	        DefProcChngOrig:
	            //================================== Traitement des reponses pour le defaut1  =============================================================//
	            IF #ChPont.Dial_Def.Reponse_Def = 'ABANDON' THEN
	                #ChPont.Dial_Def.Reponse_Def := '';
	                IF #ChPont._Commande._PtcelOrig._Moborg <> -1 AND #ChPont._Commande._PtcelOrig._Moborg <> "Index_Mobile"(#ChPont._ChargCommun.CntlDest.Dest) THEN
	                    #ChPont._ChargCommun._VidCirChgCell := TRUE;
	                END_IF;
	                #Ret_int := "RechIndexCel"(#ChPont._ChargCommun.CntlDest.Dest);
	                #ChPont._Commande._PtcelOrig := "DB_Mod_Cellule"._TabCel[#Ret_int];
	                IF #ChPont._ChargCommun._VidCirChgCell THEN
	                    #ChPont._SuspCircuit := FALSE;
	                    #ChPont._ChargCommun._CommunGeneral._Etp := #Etape_VidCircuit;
	                    RETURN;
	                ELSE
	                    #ChPont._ChargCommun._CommunGeneral._Etp := #Etape_CtrlColChute;
	                    RETURN;
	                END_IF;
	                RETURN;
	            END_IF;
	            IF #ChPont.Dial_Def.Reponse_Def = 'RELANCE' THEN
	                #ret_string := "Proc_ChangOrig"(NumPoste := "Num_Poste",
	                                                IdComLign := #ChPont._Commande._IdComLig,
	                                                IdLigOrig := #ChPont._Commande._IdLigOrig,
	                                                NvOrig := #ChPont._ChargCommun.CntlDest.Dest,
	                                                ChgAuto := 'N',
	                                                Msg_Def => #Mess_Def, ComLign := #ChPont._Commande);
	                IF #ret_string = 'NOK' THEN
	                    #ChPont.Dial_Def.Reponse_Def := '';
	                    #Text_Def := #Mess_Def;
	                    #ChPont._ParamTrouve := FALSE;
	                    #ChPont.Dial_Def.Num_Def_Etape := 3;
	                    #ChPont.Dial_Def.Index_Defaut := "Dialog_Defaut"(Fg_Base := #FgBase,
	                                                                     Msg_Defaut := #Text_Def,
	                                                                     Type_Defaut := 2,
	                                                                     Automatisme := #ChPont._ChargCommun._CommunGeneral._Autom,
	                                                                     Num_Lot := #ChPont._ChargCommun._CommunGeneral._NumLot,
	                                                                     Origine_Defaut := 'Proc Chngm Orig',
	                                                                     Libelle_Origine := 'Changement Origine',
	                                                                     Acq1 := 'ABANDON',
	                                                                     Acq2 := 'RELANCE',
	                                                                     Acq3 := '',
	                                                                     Acq4 := '',
	                                                                     Acq5 := '',
	                                                                     Acq6 := '',
	                                                                     Acq7 := '',
	                                                                     Acq8 := '',
	                                                                     Acq_Choisi := -1,
	                                                                     Date_Arrivee := #ChPont._TpsPicke);
	                    #ChPont._ChargCommun._CommunGeneral._Etp := #Etape_Attente_RepDial;
	                    RETURN;
	                ELSE
	                    IF #ChPont._Commande._PtcelOrig._Moborg <> -1 AND #ChPont._Commande._PtcelOrig._Moborg <> "Index_Mobile"(#ChPont._ChargCommun.CntlDest.Dest) THEN
	                        #ChPont._ChargCommun._VidCirChgCell := TRUE;
	                    END_IF;
	                    #Ret_int := "RechIndexCel"(#ChPont._ChargCommun.CntlDest.Dest);
	                    #ChPont._Commande._PtcelOrig := "DB_Mod_Cellule"._TabCel[#Ret_int];
	                    IF #ChPont._ChargCommun._VidCirChgCell THEN
	                        #ChPont._SuspCircuit := FALSE;
	                        #ChPont._ChargCommun._CommunGeneral._Etp := #Etape_VidCircuit;
	                        RETURN;
	                    ELSE
	                        #ChPont._ChargCommun._CommunGeneral._Etp := #Etape_CtrlColChute;
	                        RETURN;
	                    END_IF;
	                END_IF;
	            END_IF;
	            //============================================  Fin traitement  ====================================================================//







	        END_REGION Traitement cyclique "DefArrProd"
	(*
	 *************************************** *************************************** *************************************** *************************************** ***************************************
	                                                        ╔════════════════════════════════════╗
	                                                        ║          Etape "SuspChgtCase"      ║
	                                                        ╚════════════════════════════════════╝
	*************************************** *************************************** *************************************** *************************************** ***************************************
	*)
	    #Etape_SuspChgtCase:
	        REGION Traitement preliminaire "SuspChgtCase"
	            IF (#ChPont._ChargCommun._CommunGeneral._Etp <> #ChPont._ChargCommun._CommunGeneral._EtpPrec) THEN
	                #ChPont._ChargCommun._CommunGeneral._EtpPrec := #ChPont._ChargCommun._CommunGeneral._Etp;
	                #ChPont._ChargCommun._CommunGeneral._DescEtp := 'Etape SuspChgtCase';
	                "MajBtSupervChPont"(Type := 3,
	                                    ChPont := #ChPont);
	                #ChPont._MemoAppuiBP := 0;
	            END_IF;
	        END_REGION Traitement preliminaire
	        REGION Traitement cyclique "SuspChgtCase"

	            IF #ChPont._ChargDebit THEN
	                "SuspCalculDebit"(Type := "BTSUSP",
	                                  ParCal := #ChPont._ChargCommun._CommunGeneral._ParCal);
	            END_IF;
	            IF #ChPont._Commande._Case < #ChPont._Commande._NbCase - 1 AND #ChPont._DemChgtCase = 0 THEN
	                #ChPont._IndexTemp := #ChPont._Commande._Case + 1;
	                "MemoPoidsCase"(IndexNouvCase := #ChPont._IndexTemp,
	                                Chpont := #ChPont);

	            ELSIF #ChPont._DemChgtCase <> 0 THEN
	                #ChPont._IndexTemp := #ChPont._DemChgtCase;
	                "MemoPoidsCase"(IndexNouvCase := #ChPont._IndexTemp,
	                                Chpont := #ChPont);
	                #ChPont._DemChgtCase := 0;

	            ELSE
	                //Affiche mssg def: Quantite case camion atteinte, veuillez choisir une nouvelle case
	                //Selection parmi  pt_zs->Cases[i].noCase
	                ;
	            END_IF;
	            #ChPont._ChargCommun._PtAff._MessOper := 'Attente positionnement camion et DepCycle ou FinChar pour vidanger';
	            #ChPont._ChargCommun._PtAff._NumCaseEc := #ChPont._Commande._Case;
	            #ChPont._DemChgtCase := 0;
	            #ChPont._Bouton := "LireActionBoutonChPont"(#ChPont);
	            IF #ChPont._Bouton = "DEBCYCLE" THEN
	                #ChPont._BtDepCycle := 1;
	                #ChPont._MemoAppuiBP := 0;
	                IF "CondChargement"(#ChPont) AND "FC_Test_Niv_AmontAval"(Num_Zone := #ChPont._ChargCommun._CommunGeneral._NumZone, Lst_Taches := #ChPont._ListeTaAttAutDemarrage) THEN
	                    #ChPont._SuspCircuit := FALSE;
	                    IF #ChPont._ChargDebit THEN
	                        "SuspCalculDebit"(Type := "DEBCYCLE",
	                                          ParCal := #ChPont._ChargCommun._CommunGeneral._ParCal);
	                    END_IF;
	                    #ChPont._ChargCommun._CommunGeneral._Etp := #Etape_Extract;
	                    RETURN;
	                END_IF;
	            END_IF;

	            IF #ChPont._Bouton = "ABANDONCHARG" THEN
	                #ChPont._SuspCircuit := FALSE;
	                #ChPont._Ptzs._FgStopMiPesee := FALSE;
	                #ChPont._ChargCommun._CommunGeneral._Etp := #Etape_VidCircuit;
	                RETURN;
	            END_IF;
	            "ControleChgtCase"(#ChPont);



	        END_REGION Traitement cyclique "SuspChgtCase"
	    (*
	    *************************************** *************************************** *************************************** *************************************** ***************************************
	                                                        ╔════════════════════════════════════╗
	                                                        ║          Etape "SuspChargement"    ║
	                                                        ╚════════════════════════════════════╝
	    *************************************** *************************************** *************************************** *************************************** ***************************************
	    *)
	    #Etape_SuspChargement:
	        REGION Traitement preliminaire "SuspChargement"
	            IF (#ChPont._ChargCommun._CommunGeneral._Etp <> #ChPont._ChargCommun._CommunGeneral._EtpPrec) THEN
	                #ChPont._ChargCommun._CommunGeneral._EtpPrec := #ChPont._ChargCommun._CommunGeneral._Etp;
	                #ChPont._ChargCommun._CommunGeneral._DescEtp := 'Etape SuspChargement';
	                //Suspension calcul debit
	                IF #ChPont._ChargDebit THEN
	                    "SuspCalculDebit"(Type := "BTSUSP",
	                                      ParCal := #ChPont._ChargCommun._CommunGeneral._ParCal);
	                END_IF;
	                "MajBtSupervChPont"(Type := 3,
	                                    ChPont := #ChPont);
	                #ChPont._ChargCommun._PtAff._MessOper := 'Suspension chargement';
	            END_IF;
	        END_REGION Traitement preliminaire
	        REGION Traitement cyclique "SuspChargement"
	            #ChPont._Bouton := "LireActionBoutonChPont"(#ChPont);
	            IF #ChPont._Commande._FgaVider THEN
	                IF #ChPont._ChargCommun._BpVide THEN
	                    #ChPont._Ptzs._TypeArret := "ARRET_VIDE";
	                    #ChPont._AutorMAJColChute := FALSE;
	                    #ChPont._ChargCommun._CommunGeneral._Etp := #Etape_VidCircuit;
	                    RETURN;
	                END_IF;
	            END_IF;
	            IF "CondChargement"(#ChPont) AND #ChPont._Bouton = "DEBCYCLE" THEN
	                #ChPont._SuspCircuit := FALSE;
	                IF #ChPont._ChargDebit THEN
	                    "SuspCalculDebit"(Type := "DEBCYCLE",
	                                      ParCal := #ChPont._ChargCommun._CommunGeneral._ParCal);
	                END_IF;
	                #ChPont._ChargCommun._CommunGeneral._Etp := #Etape_Extract;
	                RETURN;
	            END_IF;
	            IF #ChPont._Bouton = "ABANDONCHARG" THEN
	                IF #ChPont._ArrImmMemeProd AND #ChPont._Ptzs._FgDemArrImm THEN
	                    #ChPont._SuspCircuit := FALSE;
	                    #ChPont._Ptzs._TypeArret := "ARRET_IMM";
	                ELSE
	                    #ChPont._SuspCircuit := FALSE;
	                END_IF;
	                #ChPont._Ptzs._FgStopMiPesee := FALSE;
	                #ChPont._ChargCommun._CommunGeneral._Etp := #Etape_VidCircuit;
	                RETURN;
	            END_IF;

	            // Demande de changement de case
	            IF #ChPont._DemChgtCase <> 0 THEN
	                #ChPont._DemVib := FALSE;
	                "ArretVibreur"(#ChPont._Commande._PtcelOrig);
	                #ChPont._SuspCircuit := TRUE;
	                "Arret_Ext"(ConsQte := #ChPont._Commande._ConsQteTot,
	                            Commande := #ChPont._Commande,
	                            ChargCommun := #ChPont._ChargCommun,
	                            Ptcel := #ChPont._Commande._PtcelOrig);
	                #ChPont._ChargCommun._PtAff._ExtEc := 0;
	                #ChPont._ChargCommun._CommunGeneral._Etp := #Etape_SuspChgtCase;
	                RETURN;
	            END_IF;


	        END_REGION Traitement cyclique "SuspChargement"
	    (*
	    *************************************** *************************************** *************************************** *************************************** ***************************************
	                                                        ╔════════════════════════════════════╗
	                                                        ║      Etape "ConfFinChargement"     ║
	                                                        ╚════════════════════════════════════╝
	    *************************************** *************************************** *************************************** *************************************** ***************************************
	    *)
	    #Etape_ConfFinChargement:
	        REGION Traitement preliminaire "ConfFinChargement"
	            IF (#ChPont._ChargCommun._CommunGeneral._Etp <> #ChPont._ChargCommun._CommunGeneral._EtpPrec) THEN
	                #ChPont._ChargCommun._CommunGeneral._EtpPrec := #ChPont._ChargCommun._CommunGeneral._Etp;
	                #ChPont._ChargCommun._CommunGeneral._DescEtp := 'Etape ConfFinChargement';
	                #MajNiv := "Maj_Niv"(Num_Zone := #ChPont._ChargCommun._CommunGeneral._NumZone, Num_Tache := #ChPont._ChargCommun._CommunGeneral._Tache, Niveau := "NIV_SURPONT_CONF_FIN_CHAR");
	                #ChPont._ChargCommun._DemVibrCel := FALSE;
	                "ArretVibreur"(#ChPont._Commande._PtcelOrig);
	                #ChPont._SuspCircuit := TRUE;
	                "Arret_Ext"(ConsQte := #ChPont._Commande._ConsQteTot,
	                            Commande := #ChPont._Commande,
	                            ChargCommun := #ChPont._ChargCommun,
	                            Ptcel := #ChPont._Commande._PtcelOrig);





	                // si stop mi pesee pas de confirmation fin
	                IF #ChPont._Ptzs._FgStopMiPesee THEN
	                    #ChPont._ChargCommun._CommunGeneral._Etp := #Etape_VidCircuit;
	                    RETURN;
	                END_IF;
	                "ArretCalculDebit"(#ChPont._ChargCommun._CommunGeneral._ParCal);
	                "MajBtSupervChPont"(Type := 4,
	                                    ChPont := #ChPont);
	                IF NOT #ChPont._Ptzs._HorsPont THEN
	                    #ChPont._ChargCommun._PtAff._MessOper := 'Attente Confirmation Fin Chargement ou Ajout';
	                ELSE
	                    #ChPont._ChargCommun._PtAff._MessOper := 'Attente Camion sur pont et Confirmation Fin Chargement ou Ajout';
	                END_IF;

	                #ChPont._MemoRajout := FALSE;


	            END_IF;
	        END_REGION Traitement preliminaire
	        REGION Traitement cyclique "ConfFinChargement"
	            // On controle le changement de case dans le cas o on utilisait le bouton AJOUT
	            IF #ChPont._GestQteCaseAuto AND NOT #ChPont._Ptzs._Cases[#ChPont._Commande._Case]._FgRelCharge AND #ChPont._Commande._NbCase > 1 THEN

	                IF #ChPont._Commande._PtcelOrig._FgColChuteChgtCase = 1 THEN
	                    #ChPont._ChargCommun._QteCase := #ChPont._Ptzs._Cases[#ChPont._Commande._Case]._QteDejaChargee + #ChPont._ChargCommun._Vbasc - #ChPont._Ptzs._Cases[#ChPont._Commande._Case]._Tare + #ChPont._Commande._ChuteCel;
	                ELSIF #ChPont._Commande._PtcelOrig._FgColChuteChgtCase = 2 THEN
	                    #ChPont._ChargCommun._QteCase := #ChPont._Ptzs._Cases[#ChPont._Commande._Case]._QteDejaChargee + #ChPont._ChargCommun._Vbasc - #ChPont._Ptzs._Cases[#ChPont._Commande._Case]._Tare + #ChPont._ChuteArrImm;
	                ELSE
	                    #ChPont._ChargCommun._QteCase := #ChPont._Ptzs._Cases[#ChPont._Commande._Case]._QteDejaChargee + #ChPont._ChargCommun._Vbasc - #ChPont._Ptzs._Cases[#ChPont._Commande._Case]._Tare;
	                END_IF;

	                IF #ChPont._Ptzs._Cases[#ChPont._Commande._Case]._ConsQte > 0 AND ((#ChPont._ChargCommun._QteCase > #ChPont._Ptzs._Cases[#ChPont._Commande._Case]._ConsQte + #ChPont._TolDernCase AND #ChPont._Commande._Case = #ChPont._Commande._NbCase - 1) OR
	                    (#ChPont._ChargCommun._QteCase > #ChPont._Ptzs._Cases[#ChPont._Commande._Case]._ConsQte AND #ChPont._Commande._Case <> #ChPont._Commande._NbCase - 1)) THEN

	                    #ChPont._ChargCommun._DemVibrCel := FALSE;
	                    "ArretVibreur"(#ChPont._Commande._PtcelOrig);
	                    #ChPont._SuspCircuit := TRUE;
	                    "Arret_Ext"(ConsQte := #ChPont._Commande._ConsQteTot,
	                                Commande := #ChPont._Commande,
	                                ChargCommun := #ChPont._ChargCommun,
	                                Ptcel := #ChPont._Commande._PtcelOrig);
	                    #ChPont._Ptzs._Cases[#ChPont._Commande._Case]._FgRelCharge := TRUE;
	                    #ChPont._ChargCommun._PtAff._ExtEc := 0;
	                    #ChPont._ChargCommun._CommunGeneral._Etp := #Etape_SuspChgtCase;
	                    RETURN;
	                END_IF;
	            END_IF;

	            #ChPont._Bouton := "LireActionBoutonChPont"(#ChPont);
	            IF #ChPont._Bouton = "BTAJOUT" THEN
	                #ChPont._SuspCircuit := FALSE;
	                #ChPont._MemoRajout := TRUE;
	                #ChPont._AutorMAJColChute := FALSE;
	                #ChPont._ChargCommun._CommunGeneral._Etp := #Etape_Extract;         // #Etape_Surveillance;
	                RETURN;
	            END_IF;
	            IF #ChPont._Bouton = "ABANDONCHARG" OR #ChPont._VidAuto THEN
	                // Redemarrage circuit si pas arret immdiat
	                IF #ChPont._Ptzs._TypeArret <> "ARRET_IMM" THEN
	                    #ChPont._SuspCircuit := FALSE;
	                END_IF;
	                #ChPont._ChargCommun._CommunGeneral._Etp := #Etape_VidCircuit;
	                RETURN;
	            END_IF;
	            IF #ChPont._Bouton = "BTSUSP" THEN
	                #ChPont._BtSusp := 1;
	                #ChPont._MemoAppuiBP := 0;
	                #ChPont._SuspCircuit := TRUE;
	                #Ret_RD_Sys_T := RD_SYS_T(#ChPont._DebFermExt);
	            END_IF;
	        END_REGION Traitement cyclique "ConfFinChargement"
	    (*
	    *************************************** *************************************** *************************************** *************************************** ***************************************
	                                                        ╔════════════════════════════════════╗
	                                                        ║          Etape "VidCircuit"        ║
	                                                        ╚════════════════════════════════════╝
	    *************************************** *************************************** *************************************** *************************************** ***************************************
	    *)
	    #Etape_VidCircuit:
	        REGION Traitement preliminaire "VidCircuit"
	            IF (#ChPont._ChargCommun._CommunGeneral._Etp <> #ChPont._ChargCommun._CommunGeneral._EtpPrec) THEN
	                #ChPont._ChargCommun._CommunGeneral._EtpPrec := #ChPont._ChargCommun._CommunGeneral._Etp;
	                #ChPont._ChargCommun._CommunGeneral._DescEtp := 'Etape VidCircuit';
	                #MajNiv := "Maj_Niv"(Num_Zone := #ChPont._ChargCommun._CommunGeneral._NumZone, Num_Tache := #ChPont._ChargCommun._CommunGeneral._Tache, Niveau := "NIV_SURPONT_VID_CIR");
	                #ChPont._ChargCommun._PtAff._MessOper := 'Vidange circuit';
	                "ArretCalculDebit"(#ChPont._ChargCommun._CommunGeneral._ParCal);
	                "Arret_Ext"(ConsQte := #ChPont._Commande._ConsQteTot,
	                            Commande := #ChPont._Commande,
	                            ChargCommun := #ChPont._ChargCommun,
	                            Ptcel := #ChPont._Commande._PtcelOrig);
	                // fonction utilisateur avant vidange circuit
	                IF #ChPont._ActionAvantVidangeCircuit THEN
	                    "ActionAvantVidangeCircuit"();
	                END_IF;
	                // Vidange cellule sur changement de cellule
	                (*  IF #ChPont._ChargCommun._VidCirChgCell THEN
	    #ChPont._ChargCommun._DefEvol := 0;
	    #ChPont._ChargCommun._CommunGeneral._Etp := #Etape_CtrlColChute;
	    #ChPont._ChargCommun._VidCirChgCell := FALSE;
	    RETURN;
	    END_IF; *)
	            END_IF;
	        END_REGION Traitement preliminaire
	        REGION Traitement cyclique "VidCircuit"
	            #ChPont._Bouton := "LireActionBoutonChPont"(#ChPont);
	            IF #ChPont._Bouton = "BTSUSP" THEN
	                #ChPont._BtSusp := 1;
	                #ChPont._MemoAppuiBP := 0;
	                #ChPont._SuspCircuit := TRUE;
	                #Ret_RD_Sys_T := RD_SYS_T(#ChPont._DebFermExt);
	            END_IF;

	            IF #ChPont._Bouton = "DEBCYCLE" THEN
	                #ChPont._BtDepCycle := 1;
	                #ChPont._MemoAppuiBP := 0;
	                #ChPont._SuspCircuit := FALSE;
	                #Ret_RD_Sys_T := RD_SYS_T(#ChPont._DebFermExt);
	            END_IF;


	            // Vidange cellule sur changement de cellule
	            IF #ChPont._ChargCommun._VidCirChgCell THEN
	                #ChPont._ChargCommun._DefEvol := 0;
	                #ChPont._ChargCommun._CommunGeneral._Etp := #Etape_AttFinVidCircuit;
	                RETURN;
	            END_IF;



	            // Arret produit suivant identique
	            IF #ChPont._Ptzs._TypeArret = "ARRET_IMM" AND NOT #ChPont._Ptzs._FgStopMiPesee THEN
	                #ChPont._SuspCircuit := TRUE;
	                #PtSuivCharg.ArrCirPlein := TRUE;
	                #ChPont._ChargCommun._CommunGeneral._Etp := #Etape_AttFinVidCompo;
	                RETURN;
	            ELSIF (#ChPont._Ptzs._TypeArret = "ARRET_EVOL" OR #ChPont._Ptzs._TypeArret = "ARRET_VIDE") AND NOT #ChPont._Ptzs._FgStopMiPesee THEN
	                #PtSuivCharg.ArrCirPlein := FALSE;
	                #Ret_Sint := "Arr_Imm_Circuit"(#ChPont._Circuit);
	                #Ret_Sint := "Libere_Circuit"(#ChPont._Circuit);
	                #ChPont._ChargCommun._CommunGeneral._Etp := #Etape_AttFinVidCompo;
	                RETURN;
	            ELSE
	                #PtSuivCharg.ArrCirPlein := FALSE;
	                #ChPont._ChargCommun._DefEvol := 0;
	                #ChPont._ChargCommun._CommunGeneral._Etp := #Etape_AttFinVidCircuit;
	                RETURN;
	            END_IF;



	        END_REGION Traitement cyclique "VidCircuit"
	    (*
	    *************************************** *************************************** *************************************** *************************************** ***************************************
	                                                        ╔════════════════════════════════════╗
	                                                        ║       Etape "AttFinVidCircuit"     ║
	                                                        ╚════════════════════════════════════╝
	    *************************************** *************************************** *************************************** *************************************** ***************************************
	    *)
	    #Etape_AttFinVidCircuit:
	        REGION Traitement preliminaire "AttFinVidCircuit"
	            IF (#ChPont._ChargCommun._CommunGeneral._Etp <> #ChPont._ChargCommun._CommunGeneral._EtpPrec) THEN
	                #ChPont._ChargCommun._CommunGeneral._EtpPrec := #ChPont._ChargCommun._CommunGeneral._Etp;
	                #ChPont._ChargCommun._CommunGeneral._DescEtp := 'Etape AttFinVidCircuit';
	                #ChPont._ChargCommun._PtAff._MessOper := 'Attente fin vidange Circuit';
	                "MajBtSupervChPont"(Type := 0,
	                                    ChPont := #ChPont);
	                //#Ret_Sint := "Fin_Pos_Circuit"(#ChPont._Circuit);
	            END_IF;
	        END_REGION Traitement preliminaire
	        REGION Traitement cyclique "AttFinVidCompo"
	            #Ret_Bool := "Vid_Circuit_Cycl"(#ChPont._Circuit);
	            "AffichePoids1"(
	                            ChargCommun := #ChPont._ChargCommun,
	                            Ptzs := #ChPont._Ptzs,
	                            Commande := #ChPont._Commande);
	            // IF "Test_Etat_Circuit"(Etat := "Enc_Fin_Pos", Debut := 0, CIRCUIT := #ChPont._Circuit) THEN

	            IF #Ret_Bool AND "Test_Etat_Circuit"(Etat := "Libre", Debut := 0, CIRCUIT := #ChPont._Circuit) THEN
	                #Ret_Sint := "Libere_Circuit"(#ChPont._Circuit);
	                IF #ChPont._ChargCommun._VidCirChgCell THEN
	                #Ret_int := "RechIndexCel"(#ChPont._ChargCommun.CntlDest.Dest);
	                #ChPont._Commande._PtcelOrig := "DB_Mod_Cellule"._TabCel[#Ret_int];
	                    #ChPont._ChargCommun._VidCirChgCell := FALSE;
	                    #ChPont._ChargCommun._CommunGeneral._Etp := #Etape_CtrlColChute;
	                    RETURN;
	                END_IF;

	                //  #ChPont._ChargCommun._CommunGeneral._Etp := #Etape_CtrlColChute;
	                #ChPont._ChargCommun._CommunGeneral._Etp := #Etape_AttFinVidCompo;
	                RETURN;
	            END_IF;
	        END_REGION Traitement cyclique "AttFinVidCompo"
	    (*
	    *************************************** *************************************** *************************************** *************************************** ***************************************
	                                                        ╔════════════════════════════════════╗
	                                                        ║       Etape "AttFinVidCompo"       ║
	                                                        ╚════════════════════════════════════╝
	    *************************************** *************************************** *************************************** *************************************** ***************************************
	    *)
	    #Etape_AttFinVidCompo:
	        REGION Traitement preliminaire "AttFinVidCompo"
	            IF (#ChPont._ChargCommun._CommunGeneral._Etp <> #ChPont._ChargCommun._CommunGeneral._EtpPrec) THEN
	                #ChPont._ChargCommun._CommunGeneral._EtpPrec := #ChPont._ChargCommun._CommunGeneral._Etp;
	                #ChPont._ChargCommun._CommunGeneral._DescEtp := 'Etape AttFinVidCompo';
	                #ChPont._ChargCommun._PtAff._MessOper := 'Attente fin chargement autre composant';
	                "MajBtSupervChPont"(Type := 0,
	                                    ChPont := #ChPont);
	            END_IF;
	        END_REGION Traitement preliminaire
	        REGION Traitement cyclique "AttFinVidCompo"
	            "AffichePoids1"(
	                            ChargCommun := #ChPont._ChargCommun,
	                            Ptzs := #ChPont._Ptzs,
	                            Commande := #ChPont._Commande);
	            IF "FC_Test_Niv_AmontAval"(Num_Zone := #ChPont._ChargCommun._CommunGeneral._NumZone, Lst_Taches := #ChPont._ListeTaAttFinVidCompo) THEN
	                IF #ChPont._ChargCommun._FgPresPont THEN
	                    #ChPont._ChargCommun._CommunGeneral._Etp := #Etape_AttPoidsStable;
	                ELSE

	                    #ChPont._ChargCommun._CommunGeneral._Etp := #Etape_TestTolerance;
	                END_IF;

	                RETURN;
	            END_IF;
	        END_REGION Traitement cyclique "AttFinVidCompo"
	    (*
	    *************************************** *************************************** *************************************** *************************************** ***************************************
	                                                        ╔════════════════════════════════════╗
	                                                        ║          Etape "AttPoidsStable"    ║
	                                                        ╚════════════════════════════════════╝
	    *************************************** *************************************** *************************************** *************************************** ***************************************
	    *)
	    #Etape_AttPoidsStable:
	        REGION Traitement preliminaire "AttPoidsStable"
	            IF (#ChPont._ChargCommun._CommunGeneral._Etp <> #ChPont._ChargCommun._CommunGeneral._EtpPrec) THEN
	                #ChPont._ChargCommun._CommunGeneral._EtpPrec := #ChPont._ChargCommun._CommunGeneral._Etp;
	                #ChPont._ChargCommun._CommunGeneral._DescEtp := 'Etape AttPoidsStable';
	                #ChPont._ChargCommun._PtAff._MessOper := 'Attente poids stable';
	                #Ret_RD_Sys_T := RD_SYS_T(#ChPont._DebStable);
	                #ChPont._MemoPoids := #ChPont._ChargCommun._Vbasc;
	                "MajBtSupervChPont"(Type := 0,
	                                    ChPont := #ChPont);
	            END_IF;
	        END_REGION Traitement preliminaire
	        REGION Traitement cyclique "AttPoidsStable"
	            "AffichePoids1"(
	                            ChargCommun := #ChPont._ChargCommun,
	                            Ptzs := #ChPont._Ptzs,
	                            Commande := #ChPont._Commande);
	            #Ret_Bool := "Tempo"(Duree := #ChPont._TpPoidsStab, Tps_Picke := #ChPont._DebStable, Anticip := FALSE, Tps_Passe => #Tps_Passe);
	            IF #Ret_Bool THEN
	                IF #ChPont._ChargCommun._Vbasc - #ChPont._MemoPoids > #ChPont._EcartPoidsStab THEN
	                    #Ret_RD_Sys_T := RD_SYS_T(#ChPont._DebStable);
	                    #ChPont._MemoPoids := #ChPont._ChargCommun._Vbasc;
	                ELSE
	                    #ChPont._ChargCommun._CommunGeneral._Etp := #Etape_TestTolerance;
	                    RETURN;
	                END_IF;
	            END_IF;

	        END_REGION Traitement cyclique "AttPoidsStable"
	    (*
	    *************************************** *************************************** *************************************** *************************************** ***************************************
	                                                        ╔════════════════════════════════════╗
	                                                        ║          Etape "TestTolerance"     ║
	                                                        ╚════════════════════════════════════╝
	    *************************************** *************************************** *************************************** *************************************** ***************************************
	    *)
	    #Etape_TestTolerance:
	        REGION Traitement preliminaire "TestTolerance"
	            IF (#ChPont._ChargCommun._CommunGeneral._Etp <> #ChPont._ChargCommun._CommunGeneral._EtpPrec) THEN
	                #ChPont._ChargCommun._CommunGeneral._EtpPrec := #ChPont._ChargCommun._CommunGeneral._Etp;
	                #ChPont._ChargCommun._CommunGeneral._DescEtp := 'Etape TestTolerance';
	                #ChPont._ChargCommun._PtAff._MessOper := 'Test Tolerance';
	                #MajNiv := "Maj_Niv"(Num_Zone := #ChPont._ChargCommun._CommunGeneral._NumZone, Num_Tache := #ChPont._ChargCommun._CommunGeneral._Tache, Niveau := "NIV_SURPONT_FVID_CIR");
	                #ChPont._Commande._QteBrut := #ChPont._ChargCommun._Vbasc;
	                #ChPont._Commande._QteNet := #ChPont._Commande._QteBrut - #ChPont._Commande._QteTare;


	                IF #ChPont._ChargCommun._CommunGeneral._EtpMemo = #Etape_ControleDest THEN
	                    #ChPont._ChargCommun._CommunGeneral._EtpMemo := -1;
	                    GOTO CtrlDestEtpTolerance;
	                END_IF;

	                #Ret_RD_Sys_T := RD_SYS_T(#ChPont._TpsPicke);
	                IF #ChPont.Dial_Def.Reponse_Def <> '' THEN
	                    CASE #ChPont.Dial_Def.Num_Def_Etape OF
	                        1:
	                            GOTO TESTTOL_DEF1;
	                        2:
	                            GOTO TESTTOL_DEF2;
	                        3:
	                            GOTO TESTTOL_DEF3;
	                    END_CASE;
	                END_IF;
	                //Si demande a completer deja effectuer pas de test tolerance
	                IF #ChPont._Ptzs._EtatChar = "A_COMPLETER" THEN
	                    #ChPont._ChargCommun._CommunGeneral._Etp := #Etape_FinLot;
	                    RETURN;
	                END_IF;
	            END_IF;

	        END_REGION Traitement preliminaire
	        REGION Traitement cyclique "TestTolerance"
	            "AffichePoids1"(
	                            ChargCommun := #ChPont._ChargCommun,
	                            Ptzs := #ChPont._Ptzs,
	                            Commande := #ChPont._Commande);
	            //Arret mi pesee pour calcul colonne de chute
	            IF #ChPont._Ptzs._FgStopMiPesee AND NOT #ChPont._Ptzs._Abandon THEN
	                #ChPont._Commande._ChuteCel := #ChPont._Commande._QteNet - #ChPont._Commande._ConsArret;
	                #ChPont._Ptzs._FgStopMiPesee := FALSE;
	                #ChPont._Ptzs._FgRelSansConf := TRUE;
	    (* "Min_Max"(Min := #ChPont._MinChute,
	         Max := #ChPont._MaxChute,
	         Val_Calc:=#ChPont._Commande._ChuteCel,
	         Sort_Ana:=#ChPont._Commande._ChuteCel); *)
	                IF #FgBase THEN
	                    //MajColChute(pt_compo, UnicodeString(WLireNomCharg()).c_str());
	                    ;
	                END_IF;
	                #ChPont._ChargCommun._CommunGeneral._Etp := #Etape_CtrlColChute;
	                RETURN;
	            ELSIF #ChPont._Commande._QteNet > (#ChPont._Commande._ConsQteTot + #ChPont._Ptzs._TolSup) AND #ChPont._ChargCommun._FgPresPont THEN
	                // Hors tolerance superieure
	                #ChPont.Dial_Def.Num_Def_Etape := 1;
	                // #reel := #ChPont._Commande._QteDejaChargee + #ChPont._Commande._QteNet;
	                // #Ecart := #ChPont._Commande._QteNet - #ChPont._Commande._ConsQte;
	                "Real_Strg"("Real" := #ChPont._Commande._ConsQteTot,
	                            Size := 5,
	                            NmbDecimal := 0,
	                            "String" => #tempConsQte);
	                "Real_Strg"("Real" := #ChPont._Commande._QteDejaCharg + #ChPont._Commande._QteNet,
	                            Size := 5,
	                            NmbDecimal := 0,
	                            "String" => #tempqtereel);
	                "Real_Strg"("Real" := #ChPont._Commande._QteNet - #ChPont._Commande._ConsQteTot,
	                            Size := 5,
	                            NmbDecimal := 0,
	                            "String" => #tempecart);
	                "Real_Strg"("Real" := #ChPont._Ptzs._TolSup,
	                            Size := 5,
	                            NmbDecimal := 0,
	                            "String" => #tolsup);

	                #Text_Def := CONCAT(IN1 := 'Defaut hors tolerance superieur ', IN2 := #ChPont._Commande._PtcelOrig._Cel, IN3 := ' Prevu:', IN4 := #tempConsQte, IN5 := ' , reel:', IN6 := #tempqtereel, IN7 := ' , Ecart:', IN8 := #tempecart, IN9 := ' , Ecart Tolere:', IN10 := #tolsup);
	                #ChPont.Dial_Def.Index_Defaut := "Dialog_Defaut"(Fg_Base := #FgBase, Msg_Defaut := #Text_Def,
	                                                                 Type_Defaut := 2,
	                                                                 Automatisme := #ChPont._ChargCommun._CommunGeneral._Autom,
	                                                                 Num_Lot := #ChPont._Commande._NoLot,
	                                                                 Origine_Defaut := 'Hors Tolerance',
	                                                                 Libelle_Origine := 'Hors Tolerance',
	                                                                 Acq1 := 'Abandon',
	                                                                 Acq2 := '',
	                                                                 Acq3 := '',
	                                                                 Acq4 := '',
	                                                                 Acq5 := '',
	                                                                 Acq6 := '',
	                                                                 Acq7 := '',
	                                                                 Acq8 := '',
	                                                                 Acq_Choisi := -1,
	                                                                 Date_Arrivee := #ChPont._TpsPicke);
	                #ChPont._ChargCommun._CommunGeneral._Etp := #Etape_Attente_RepDial;
	                RETURN;

	            ELSIF #ChPont._Commande._QteNet < (#ChPont._Commande._ConsQteTot - #ChPont._Ptzs._TolInf) AND #ChPont._ChargCommun._FgPresPont THEN
	                // Hors tolerance inferieur
	                IF #ChPont._Ptzs._EtatChar = "A_COMPLETER" THEN
	                    #ChPont._ChargCommun._CommunGeneral._Etp := #Etape_FinLot;
	                    RETURN;
	                END_IF;
	                // Si relance auto paramtr et arret sur quantit on fait une relance automatique du circuit
	                IF #ChPont._NbRelAuto > #ChPont._NbRelAutoExp AND #ChPont._Ptzs._TypeArret = "ARRET_QTE" THEN
	                    #ChPont._NbRelAuto := 0;
	                    #ChPont._ChargCommun._CommunGeneral._Etp := #Etape_RechCirc;
	                    RETURN;
	                END_IF;
	                #ChPont.Dial_Def.Num_Def_Etape := 2;
	                "Real_Strg"("Real" := #ChPont._Commande._ConsQteTot,
	                            Size := 5,
	                            NmbDecimal := 0,
	                            "String" => #tempConsQte);
	                "Real_Strg"("Real" := #ChPont._Commande._QteDejaCharg + #ChPont._Commande._QteNet,
	                            Size := 5,
	                            NmbDecimal := 0,
	                            "String" => #tempqtereel);
	                "Real_Strg"("Real" := #ChPont._Commande._ConsQteTot - #ChPont._Commande._QteNet,
	                            Size := 5,
	                            NmbDecimal := 0,
	                            "String" => #tempecart);
	                "Real_Strg"("Real" := #ChPont._Ptzs._TolInf,
	                            Size := 5,
	                            NmbDecimal := 0,
	                            "String" => #tolinf);
	                #Text_Def := CONCAT(IN1 := 'Defaut hors tolerance inferieure ', IN2 := #ChPont._Commande._PtcelOrig._Cel, IN3 := ' Prevu:', IN4 := #tempConsQte, IN5 := ' , reel:', IN6 := #tempqtereel, IN7 := ' , Ecart:', IN8 := #tempecart, IN9 := ' , Ecart Tolere:', IN10 := #tolinf);
	                #ChPont.Dial_Def.Index_Defaut := "Dialog_Defaut"(Fg_Base := #FgBase, Msg_Defaut := #Text_Def,
	                                                                 Type_Defaut := 2,
	                                                                 Automatisme := #ChPont._ChargCommun._CommunGeneral._Autom,
	                                                                 Num_Lot := #ChPont._Commande._NoLot,
	                                                                 Origine_Defaut := 'Hors Tolerance',
	                                                                 Libelle_Origine := 'Hors Tolerance',
	                                                                 Acq1 := 'Relance',
	                                                                 Acq2 := 'Abandon',
	                                                                 Acq3 := 'Cellule',
	                                                                 Acq4 := 'Completer',
	                                                                 Acq5 := '',
	                                                                 Acq6 := '',
	                                                                 Acq7 := '',
	                                                                 Acq8 := '',
	                                                                 Acq_Choisi := -1,
	                                                                 Date_Arrivee := #ChPont._TpsPicke);
	                #ChPont._ChargCommun._CommunGeneral._Etp := #Etape_Attente_RepDial;
	                RETURN;
	            ELSE
	                #ChPont._Ptzs._EtatChar := "FIN_CHARG";
	                #ChPont._ChargCommun._CommunGeneral._Etp := #Etape_FinLot;
	                RETURN;
	            END_IF;
	        TESTTOL_DEF1:
	            //============ Traitement des reponses pour le defaut Hors tolerance superieur  ====================================//
	            IF #ChPont.Dial_Def.Reponse_Def = 'Abandon' THEN
	                #ChPont.Dial_Def.Reponse_Def := '';
	                #ChPont._Ptzs._Abandon := TRUE;
	                #ChPont._Ptzs._EtatChar := "FIN_CHARG";
	                #ChPont._ChargCommun._CommunGeneral._Etp := #Etape_FinLot;
	                RETURN;
	            END_IF;
	            //============ Fin Traitement des reponses pour le defaut Hors tolerance superieur  ====================================//


	        TESTTOL_DEF2:
	            //============ Traitement des reponses pour le defaut Hors tolerance inferieur  ====================================//
	            IF #ChPont.Dial_Def.Reponse_Def = 'Relance' THEN
	                #ChPont._Ptzs._Abandon := FALSE;
	                #ChPont._Ptzs._FgRelSansConf := TRUE;
	                #ChPont.Dial_Def.Reponse_Def := '';
	                IF #ChPont._Commande._ChuteCel > #ChPont._Commande._QteNet - #ChPont._Commande._ConsQteTot THEN
	                    // Calc_Temps_Relance(Comm_Ec,Pont);
	                    ;
	                END_IF;
	                IF #ChPont._Ptzs._HorsPont AND #ChPont._ChargTelem THEN
	                    #ChPont._ChargCommun._CommunGeneral._Etp := #Etape_AttCond;
	                    RETURN;
	                ELSE
	                    #ChPont._ChargCommun._CommunGeneral._Etp := #Etape_CtrlColChute;
	                    RETURN;
	                END_IF;
	            END_IF;
	            IF #ChPont.Dial_Def.Reponse_Def = 'Abandon' THEN
	                #ChPont.Dial_Def.Num_Def_Etape := 3;
	                #ChPont.Dial_Def.Reponse_Def := '';
	                #ChPont.Dial_Def.Index_Defaut := "Dialog_Defaut"(Fg_Base := #FgBase,
	                                                                 Msg_Defaut := 'Voulez vous reellement cloturer la commande',
	                                                                 Type_Defaut := 2,
	                                                                 Automatisme := #ChPont._ChargCommun._CommunGeneral._Autom,
	                                                                 Num_Lot := #ChPont._Commande._NoLot,
	                                                                 Origine_Defaut := 'Abandon de la commande',
	                                                                 Libelle_Origine := 'Abandon de la commande',
	                                                                 Acq1 := 'Oui',
	                                                                 Acq2 := 'Non',
	                                                                 Acq3 := '',
	                                                                 Acq4 := '',
	                                                                 Acq5 := '',
	                                                                 Acq6 := '',
	                                                                 Acq7 := '',
	                                                                 Acq8 := '',
	                                                                 Acq_Choisi := -1,
	                                                                 Date_Arrivee := #ChPont._TpsPicke);
	                #ChPont._ChargCommun._CommunGeneral._Etp := #Etape_Attente_RepDial;
	                RETURN;
	            END_IF;
	            IF #ChPont.Dial_Def.Reponse_Def = 'Completer' THEN
	                #ChPont.Dial_Def.Reponse_Def := '';
	                #ChPont._Ptzs._EtatChar := "A_COMPLETER";
	                #ChPont._ChargCommun._CommunGeneral._Etp := #Etape_FinLot;
	                RETURN;
	            END_IF;
	            IF #ChPont.Dial_Def.Reponse_Def = 'Cellule' THEN
	                #ChPont.Dial_Def.Reponse_Def := '';
	                #ChPont._ChargCommun.CntlDest.Dest := #ChPont.Dial_Def.Text_Reponse;
	                #ChPont._ChargCommun._CommunGeneral._Etp := #Etape_ControleDest;
	                RETURN;
	            END_IF;
	    (* #CelVid := '?';
	    "CtrlDest_1"(fgbase := #FgBase,
	         ChComm := #ChPont._ChargCommun,
	         Dial_Def := #ChPont.Dial_Def,
	         PtComp := #ChPont._Commande,
	         CdMat := #ChPont._Commande._CdMat,
	         Cel := "DB_Mod_Cellule",
	         CelVid := #CelVid); *)
	         //============ Fin  Traitement des reponses pour le defaut Hors tolerance inferieur  ====================================//







	     TESTTOL_DEF3:
	         //============ Traitement des reponses pour le defaut Confirmation d'abandon ====================================//
	         IF #ChPont.Dial_Def.Reponse_Def = 'Oui' THEN
	             #ChPont.Dial_Def.Reponse_Def := '';
	             #ChPont._Ptzs._EtatChar := "FIN_CHARG";
	             #ChPont._ChargCommun._CommunGeneral._Etp := #Etape_FinLot;
	             RETURN;
	         END_IF;
	         IF #ChPont.Dial_Def.Reponse_Def = 'Non' THEN
	             #ChPont.Dial_Def.Reponse_Def := '';
	             #ChPont._ChargCommun._CommunGeneral._Etp := #Etape_TestTolerance;
	             RETURN;
	         END_IF;


	     CtrlDestEtpTolerance:
	         IF #ChPont._ChargCommun.CntlDest.TestComplet THEN
	             IF #ChPont._ChargCommun.CntlDest.Controle = #Abandon OR #ChPont._ChargCommun.CntlDest.Controle = #AutrePont THEN
	                 IF #ChPont._ChargCommun.CntlDest.Controle = #AutrePont THEN
	                     #ChPont._Ptzs._AutrePont := TRUE;
	                 END_IF;
	                 #ChPont._Ptzs._EtatChar := "A_COMPLETER"; //A completer
	                 #ChPont._ChargCommun._CommunGeneral._Etp := #Etape_FinLot;
	                 #ChPont.Dial_Def.Reponse_Def := '';
	                 #ChPont._Ptzs._Abandon := TRUE;
	                 RETURN;
	             END_IF;

	             IF #ChPont._ChargCommun.CntlDest.Controle = #TestValide THEN

	                 #ChPont.Dial_Def.Reponse_Def := '';
	                 IF #ChPont._Commande._PtcelOrig._Moborg <> -1 AND #ChPont._Commande._PtcelOrig._Moborg <> "Index_Mobile"(#ChPont._ChargCommun.CntlDest.Dest) THEN
	                     #ChPont._ChargCommun._VidCirChgCell := TRUE;
	                 END_IF;
	                 #Ret_int := "RechIndexCel"(#ChPont._ChargCommun.CntlDest.Dest);
	                 #ChPont._Commande._PtcelOrig := "DB_Mod_Cellule"._TabCel[#Ret_int];

	                 IF #ChPont._ChargCommun._VidCirChgCell THEN
	                     #ChPont._SuspCircuit := FALSE;
	                     #ChPont._ChargCommun._CommunGeneral._Etp := #Etape_VidCircuit;
	                     RETURN;
	                 ELSE
	                     #ChPont._ChargCommun._CommunGeneral._Etp := #Etape_CtrlColChute;
	                     RETURN;
	                 END_IF;
	             END_IF;
	         END_IF;



	     END_REGION Traitement cyclique "TestTolerance"
	     (*
	     *************************************** *************************************** *************************************** *************************************** ***************************************
	                                                                     ╔════════════════════════════════════╗
	                                                                     ║          Etape "FinLot"            ║
	                                                                     ╚════════════════════════════════════╝
	     *************************************** *************************************** *************************************** *************************************** ***************************************
	     *)
	    #Etape_FinLot:
	     REGION Traitement preliminaire "FinLot"
	         IF (#ChPont._ChargCommun._CommunGeneral._Etp <> #ChPont._ChargCommun._CommunGeneral._EtpPrec) THEN
	             #ChPont._ChargCommun._CommunGeneral._EtpPrec := #ChPont._ChargCommun._CommunGeneral._Etp;
	             #ChPont._ChargCommun._CommunGeneral._DescEtp := 'Etape FinLot';
	             #ChPont._ChargCommun._PtAff._MessOper := 'Controle poids';
	             #MajNiv := "Maj_Niv"(Num_Zone := #ChPont._ChargCommun._CommunGeneral._NumZone, Num_Tache := #ChPont._ChargCommun._CommunGeneral._Tache, Niveau := "NIV_SURPONT_ATT_FINLOT");
	             "SuspCalculDebit"(Type := "BTSUSP",
	                               ParCal := #ChPont._ChargCommun._CommunGeneral._ParCal);
	             #ChPont._ChargCommun._PtAff.CompoComEc[#ChPont._ChargCommun._PtAff._NumCompoEc]._FgChrgEnc := 2;
	             #Ret_RD_Sys_T := RD_SYS_T(#ChPont._TpsPicke);
	             IF #ChPont.Dial_Def.Reponse_Def <> '' THEN
	                 CASE #ChPont.Dial_Def.Num_Def_Etape OF
	                     1:
	                         GOTO Def_UpdateStock;
	                     2:
	                         GOTO Def_FinLigCom;
	                     3:
	                         GOTO Def_FinTour;

	                 END_CASE;
	             END_IF;

	         END_IF;
	     END_REGION Traitement preliminaire
	     REGION Traitement cyclique "FinLot"
	         IF NOT "FC_Test_Niv_AmontAval"(Num_Zone := #ChPont._ChargCommun._CommunGeneral._NumZone, Lst_Taches := #ChPont._ListeTaAttFinCharg) THEN
	             RETURN;
	         END_IF;
	             IF NOT #ChPont._Ptzs._Abandon THEN
	                 // Prise poids brut
	                 IF #ChPont._Ptzs._HorsPont = FALSE THEN
	                     ;
	                     (* IF NOT  (!Poids_DSD(pt_zs, BRUT) THEN
	                          RETURN ;
	                      END_IF; *)
	                 END_IF;
	                 // Mise a jour colonne de chute
	                 IF #ChPont._ChargCommun._ValidCorColChute AND #ChPont._AutorMAJColChute THEN
	                     // Controle de la correction maximum de la colonne de chute
	                     #TempDbl := #ChPont._Commande._QteBrut - #ChPont._Commande._QteTare - #ChPont._Commande._ConsArret;
	                     IF #TempDbl > #ChPont._Commande._ChuteCel + #ChPont._ChargCommun._CorMaxColChute THEN
	                         #ChPont._Commande._ChuteCel := #ChPont._Commande._ChuteCel + #ChPont._ChargCommun._CorMaxColChute;
	                     ELSIF #TempDbl < #ChPont._Commande._ChuteCel - #ChPont._ChargCommun._CorMaxColChute THEN
	                         #ChPont._Commande._ChuteCel := #ChPont._Commande._ChuteCel - #ChPont._ChargCommun._CorMaxColChute;
	                     ELSE
	                         #ChPont._Commande._ChuteCel := #TempDbl;
	                     END_IF;
	                     "Min_Max"(Min := #ChPont._MinChute,
	                               Max := #ChPont._MaxChute,
	                               Val_Calc := #ChPont._Commande._ChuteCel,
	                               Sort_Ana := #ChPont._Commande._ChuteCel);
	                     IF #FgBase THEN
	                         ;
	                         //MajColChute(pt_compo, UnicodeString(WLireNomCharg()).c_str());;
	                     END_IF;
	                 ELSE
	                     IF #FgBase THEN
	                         ;




	                     END_IF;
	                 END_IF;

	             END_IF;
	             #ChPont._ChargCommun._PtAff.CompoComEc[#ChPont._Ptzs._NumCommande]._FgChrgEnc := 2;

	             // Appel Proc Update Stock
	         AppelProcUpdate:
	             #ChPont._Commande._QteChOrig := #ChPont._ChargCommun._Vbasc - #ChPont._Commande._QteTare - #ChPont._Commande._QteChOrig;
	             IF #FgBase THEN
	                 (* IF #ChPont._Commande._QteChOrig > 0 THEN
	                     #ChPont._Commande._TareCel := #ChPont._ChargCommun._Vbasc - (#ChPont._Commande._QteChOrig + #ChPont._Commande._QteNet);
	                 END_IF; *)
	                 IF #ChPont._Commande._TareCel > 0 THEN
	                     #ret_string := "Proc_MajStock"(ChPont := #ChPont,
	                                                    Typemouvement := '010',
	                                                    Err_Sql => #Err_Sql,
	                                                    Msg_Def => #Mess_Def);
	                     #Commande._TareCel := #ChPont._ChargCommun._Vbasc;
	                 END_IF;
	                 IF #ret_string = 'NOK' THEN
	                     #Text_Def := #Mess_Def;
	                     #ChPont._ParamTrouve := FALSE;
	                     #ChPont.Dial_Def.Num_Def_Etape := 1;
	                     #ChPont.Dial_Def.Index_Defaut := "Dialog_Defaut"(Fg_Base := #FgBase,
	                                                                      Msg_Defaut := #Text_Def,
	                                                                      Type_Defaut := 2,
	                                                                      Automatisme := #ChPont._ChargCommun._CommunGeneral._Autom,
	                                                                      Num_Lot := #ChPont._ChargCommun._CommunGeneral._NumLot,
	                                                                      Origine_Defaut := 'Update Stock',
	                                                                      Libelle_Origine := 'BD FinLot',
	                                                                      Acq1 := 'ABANDON',
	                                                                      Acq2 := 'RELANCE',
	                                                                      Acq3 := '',
	                                                                      Acq4 := '',
	                                                                      Acq5 := '',
	                                                                      Acq6 := '',
	                                                                      Acq7 := '',
	                                                                      Acq8 := '',
	                                                                      Acq_Choisi := -1,
	                                                                      Date_Arrivee := #ChPont._TpsPicke);
	                     #ChPont._ChargCommun._CommunGeneral._Etp := #Etape_Attente_RepDial;
	                     RETURN;
	                 END_IF;
	             END_IF;

	             AppelProcFinLigCom:
	             IF #FgBase THEN
	                 IF #ChPont._Ptzs._EtatChar = "A_COMPLETER" THEN
	                     #Etat := "A_COMPLETER";//c
	                 ELSE
	                     #Etat := 'T';
	                 END_IF;
	                 #ret_string := "Proc_FinComm"(NumPoste := "Num_Poste",
	                                               IdComLign := #ChPont._Commande._IdComLig,
	                                               Etat := #Etat,
	                                               Msg_Def => #Mess_Def);
	                 IF #ret_string = 'NOK' THEN
	                     #Text_Def := #Mess_Def;
	                     #ChPont._ParamTrouve := FALSE;
	                     #ChPont.Dial_Def.Num_Def_Etape := 2;
	                     #ChPont.Dial_Def.Index_Defaut := "Dialog_Defaut"(Fg_Base := #FgBase,
	                                                                      Msg_Defaut := #Text_Def,
	                                                                      Type_Defaut := 2,
	                                                                      Automatisme := #ChPont._ChargCommun._CommunGeneral._Autom,
	                                                                      Num_Lot := #ChPont._ChargCommun._CommunGeneral._NumLot,
	                                                                      Origine_Defaut := 'Fin LigComm',
	                                                                      Libelle_Origine := 'BD FinLot',
	                                                                      Acq1 := 'ABANDON',
	                                                                      Acq2 := 'RELANCE',
	                                                                      Acq3 := '',
	                                                                      Acq4 := '',
	                                                                      Acq5 := '',
	                                                                      Acq6 := '',
	                                                                      Acq7 := '',
	                                                                      Acq8 := '',
	                                                                      Acq_Choisi := -1,
	                                                                      Date_Arrivee := #ChPont._TpsPicke);
	                     #ChPont._ChargCommun._CommunGeneral._Etp := #Etape_Attente_RepDial;
	                     RETURN;
	                 END_IF;
	             END_IF;

	             AppelProcFinTour:
	             #ChPont._Commande := #Commande;
	             #ChPont._ChargCommun._CommunGeneral._ParCal := #ParCal;
	             #ChPont._Ptzs._TareOk := 0;
	             #ChPont._Ptzs._FgStopMiPesee := FALSE;
	             #ChPont._ChargCommun._CommunGeneral._Etp := #Etape_Repos;
	             #ChPont._Ptzs._NumCommande := #ChPont._Ptzs._NumCommande + 1;
	             IF #ChPont._Ptzs._NumCommande >= #ChPont._Ptzs._NbCommande THEN
	                 #ChPont._ChargCommun._PtAff._MessOper := CONCAT(IN1 := 'Fin des commandes de la tournee', IN2 := #ChPont._ChargCommun._PtAff.Tournee._CdTour);
	                 IF #ChPont.Dial_Def.Reponse_Def <> 'ABANDON' THEN
	                     #ret_string := "Proc_FinTour"(NumPoste := "Num_Poste",
	                                                   IdTourn := #ChPont._Ptzs._InfoTour._IdTourn,
	                                                   Msg_Def => #Mess_Def);
	                 END_IF;

	               IF #ret_string = 'NOK' THEN
	                   #Text_Def := #Mess_Def;
	                   #ChPont._ParamTrouve := FALSE;
	                   #ChPont.Dial_Def.Num_Def_Etape := 3;
	                   #ChPont.Dial_Def.Index_Defaut := "Dialog_Defaut"(Fg_Base := #FgBase,
	                                                                    Msg_Defaut := #Text_Def,
	                                                                    Type_Defaut := 2,
	                                                                    Automatisme := #ChPont._ChargCommun._CommunGeneral._Autom,
	                                                                    Num_Lot := #ChPont._ChargCommun._CommunGeneral._NumLot,
	                                                                    Origine_Defaut := 'Update Stock',
	                                                                    Libelle_Origine := 'BD FinLot',
	                                                                    Acq1 := 'ABANDON',
	                                                                    Acq2 := 'RELANCE',
	                                                                    Acq3 := '',
	                                                                    Acq4 := '',
	                                                                    Acq5 := '',
	                                                                    Acq6 := '',
	                                                                    Acq7 := '',
	                                                                    Acq8 := '',
	                                                                    Acq_Choisi := -1,
	                                                                    Date_Arrivee := #ChPont._TpsPicke);
	                   #ChPont._ChargCommun._CommunGeneral._Etp := #Etape_Attente_RepDial;
	                   RETURN;
	               END_IF;
	               #ChPont.Dial_Def.Reponse_Def := '';
	                 #MajNiv := "Maj_Niv"(Num_Zone := #ChPont._ChargCommun._CommunGeneral._NumZone, Num_Tache := #ChPont._ChargCommun._CommunGeneral._Tache, Niveau := "N_FINLOT");
	                 #Ret_Sint := "Libere_Zone_Suiv_Lot"(#ChPont._ChargCommun._CommunGeneral._NumZone);
	                 FOR #i := 0 TO #ChPont._Ptzs._NbCommande DO
	                     #ChPont._ChargCommun._PtAff.CompoComEc[#i]._FgChrgEnc := 0;
	                 END_FOR;

	                 #ChPont._Commande := #Commande;
	                 #ChPont._Ptzs := #Ptzs;
	                 (* "AffichePoids_1"(ChargCommun := #ChPont._ChargCommun,
	                                  Ptzs := #ChPont._Ptzs,
	                                  PtCompo := #ChPont._Commande); *)
	                 "InitTableComp"(ChargCommun := #ChPont._ChargCommun,
	                                 Ptzs := #ChPont._Ptzs,
	                                 Commande := #ChPont._Commande);
	                 #ChPont._ChargCommun._CommunGeneral._Etp := #Etape_Repos;

	                 RETURN;
	             END_IF;
	             RETURN;


	     Def_UpdateStock:
	         //================================== Traitement des reponses pour le defaut1  =============================================================//
	         IF #ChPont.Dial_Def.Reponse_Def = 'ABANDON' THEN
	             #ChPont.Dial_Def.Reponse_Def := '';
	             GOTO AppelProcFinLigCom;
	         END_IF;
	         IF #ChPont.Dial_Def.Reponse_Def = 'RELANCE' THEN
	             #ChPont.Dial_Def.Reponse_Def := '';
	             GOTO AppelProcUpdate;
	         END_IF;
	         //============================================  Fin traitement  ====================================================================//

	         Def_FinLigCom:
	         //================================== Traitement des reponses pour le defaut1  =============================================================//
	         IF #ChPont.Dial_Def.Reponse_Def = 'ABANDON' THEN
	             #ChPont.Dial_Def.Reponse_Def := '';
	             GOTO AppelProcFinTour;
	         END_IF;
	         IF #ChPont.Dial_Def.Reponse_Def = 'RELANCE' THEN
	             #ChPont.Dial_Def.Reponse_Def := '';
	             GOTO AppelProcFinLigCom;
	         END_IF;
	         //============================================  Fin traitement  ====================================================================//


	     Def_FinTour:
	         //================================== Traitement des reponses pour le defaut1  =============================================================//
	         IF #ChPont.Dial_Def.Reponse_Def = 'ABANDON' THEN
	             #ChPont._Ptzs._NumCommande := #ChPont._Ptzs._NumCommande - 1;
	             GOTO AppelProcFinTour;
	         END_IF;
	         IF #ChPont.Dial_Def.Reponse_Def = 'RELANCE' THEN
	             #ChPont.Dial_Def.Reponse_Def := '';
	             #ChPont._Ptzs._NumCommande := #ChPont._Ptzs._NumCommande - 1;
	             GOTO AppelProcFinTour;
	         END_IF;
	         //============================================  Fin traitement  ====================================================================//


	     END_REGION Traitement cyclique "FinLot"

	     (*
	     *************************************** *************************************** *************************************** *************************************** *************************************** ***************************************
	                                                                                 ╔════════════════════════════════════╗
	                                                                                 ║ Etape "Attente Reponse Dialogue"   ║
	                                                                                 ╚════════════════════════════════════╝
	     *************************************** *************************************** *************************************** *************************************** *************************************** ***************************************
	     *)
	    #Etape_Attente_RepDial:
	     REGION Preliminaire Attente Acquuitement
	         IF #ChPont._ChargCommun._CommunGeneral._Etp <> #ChPont._ChargCommun._CommunGeneral._EtpPrec THEN
	             //Memorisation de l'etape encours
	             #ChPont._ChargCommun._CommunGeneral._EtpMemo := #ChPont._ChargCommun._CommunGeneral._EtpPrec;

	             #ChPont._ChargCommun._CommunGeneral._DescEtp := 'Etape_Attente_RepDial';
	             #ChPont._ChargCommun._CommunGeneral._EtpPrec := #ChPont._ChargCommun._CommunGeneral._Etp;

	         END_IF;
	     END_REGION Preliminaire Attente Acquuitement
	     REGION Cyclique Attente Acquitement
	         #ChPont.Dial_Def.Reponse_Def := "FC_Recup_Rep_Def"(Index_Def := #ChPont.Dial_Def.Index_Defaut, Reponse_Ecrit => #ChPont.Dial_Def.Text_Reponse);
	         IF #ChPont.Dial_Def.Reponse_Def <> '' THEN
	             "FC_Raz_Def"(#ChPont.Dial_Def.Index_Defaut);
	             #ChPont._ChargCommun._CommunGeneral._Etp := #ChPont._ChargCommun._CommunGeneral._EtpMemo;
	             RETURN;
	         END_IF;
	     END_REGION Cyclique Attente Acquitement

	    (*
	    *************************************** *************************************** *************************************** *************************************** *************************************** ***************************************
	                                                                           ╔════════════════════════════════════╗
	                                                                           ║         Etape "ControleDest"       ║
	                                                                           ╚════════════════════════════════════╝
	    *************************************** *************************************** *************************************** *************************************** *************************************** ***************************************
	    *)
	    #Etape_ControleDest:
	     REGION Preliminaire
	         IF #ChPont._ChargCommun._CommunGeneral._Etp <> #ChPont._ChargCommun._CommunGeneral._EtpPrec THEN
	             //Memorisation de l'etape encours
	             #ChPont._ChargCommun._CommunGeneral._EtpMemo := #ChPont._ChargCommun._CommunGeneral._EtpPrec;

	             #ChPont._ChargCommun._CommunGeneral._DescEtp := 'Etape_ControleDest';
	             #ChPont._ChargCommun._CommunGeneral._EtpPrec := #ChPont._ChargCommun._CommunGeneral._Etp;

	         END_IF;
	     END_REGION Preliminaire
	     REGION Cyclique Attente Acquitement
	         "AffichePoids1"(
	                         ChargCommun := #ChPont._ChargCommun,
	                         Ptzs := #ChPont._Ptzs,
	                         Commande := #ChPont._Commande);
	         "CtrlDest"(fgbase := #FgBase,
	                    ChComm := #ChPont._ChargCommun,
	                    Dial_Def := #ChPont.Dial_Def,
	                    Commande := #ChPont._Commande,
	                    CdMat := #ChPont._Commande._CdMat,
	                    Cel := "DB_Mod_Cellule",
	                    CelVid := #CelVid);


	         IF #ChPont._ChargCommun.CntlDest.TestComplet THEN

	             #ChPont._ChargCommun._CommunGeneral._Etp := #ChPont._ChargCommun._CommunGeneral._EtpMemo;
	             #ChPont._ChargCommun._CommunGeneral._EtpMemo := #ChPont._ChargCommun._CommunGeneral._EtpPrec;
	         END_IF;

	     END_REGION Cyclique Attente Acquitement


	    END_CASE;
END_FUNCTION

